ABB RAPID module: Module1.mod

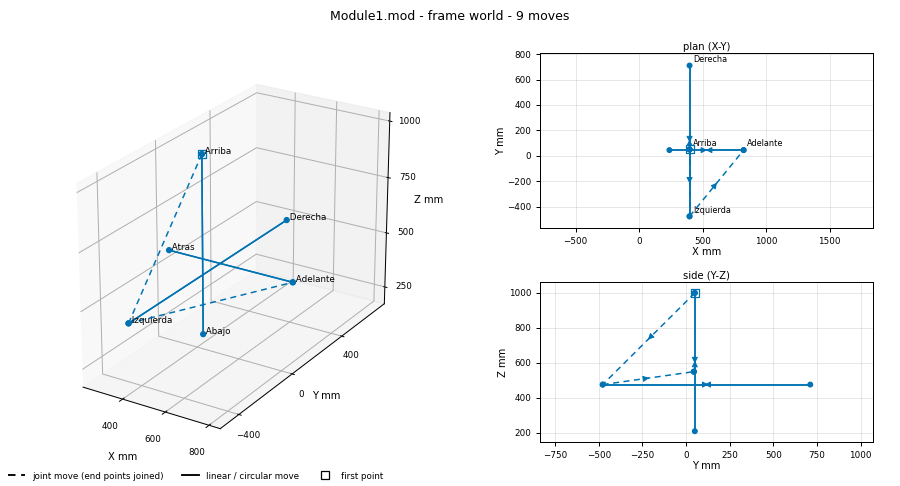
[picture p0: tool path of Module1.mod in frame world, 9 of 9 moves have a stored position in this frame; points joined in program order, loops and branches not executed]
MODULE Module1
        CONST robtarget Target_10:=[[397.237396506,49.895027971,999.967806709],[0.500000144,-0.000000762,0.86602532,-0.000000259],[0,-1,0,0],[9E+09,9E+09,9E+09,9E+09,9E+09,9E+09]];
    CONST robtarget Target_20:=[[397.2373779,49.895029997,208.416392869],[0.500000126,-0.000000768,0.866025331,-0.000000222],[0,-2,1,0],[9E+09,9E+09,9E+09,9E+09,9E+09,9E+09]];
    CONST robtarget Target_30:=[[823.141261344,44.509056663,549.297530143],[0.500000173,-0.000000339,0.866025304,-0.000000462],[0,1,-2,1],[9E+09,9E+09,9E+09,9E+09,9E+09,9E+09]];
    CONST robtarget Target_40:=[[238.396814188,44.509066911,549.297510446],[0.500000164,-0.000000322,0.866025309,-0.000000435],[0,1,-2,1],[9E+09,9E+09,9E+09,9E+09,9E+09,9E+09]];
    CONST robtarget Target_50:=[[397.237392628,-293.472887343,485.395595719],[0.500000125,-0.000000729,0.866025331,-0.000000243],[-1,0,-2,0],[9E+09,9E+09,9E+09,9E+09,9E+09,9E+09]];
    CONST robtarget Target_60:=[[397.237393587,50.453069476,485.39558546],[0.500000114,-0.000000756,0.866025338,-0.000000264],[0,1,-1,1],[9E+09,9E+09,9E+09,9E+09,9E+09,9E+09]];
    CONST robtarget Target_70:=[[802.304016355,50.453065947,615.789609831],[0.500000141,-0.000000543,0.866025322,-0.000000186],[0,1,-2,1],[9E+09,9E+09,9E+09,9E+09,9E+09,9E+09]];
    CONST robtarget Target_80:=[[271.909522335,50.453072281,615.789590887],[0.500000145,-0.000000573,0.86602532,-0.000000214],[0,1,-2,1],[9E+09,9E+09,9E+09,9E+09,9E+09,9E+09]];
    CONST robtarget Izquierda:=[[397.237378301,-477.405403417,475.381603255],[0.500000116,-0.000000746,0.866025337,-0.000000266],[-1,-2,0,1],[9E+09,9E+09,9E+09,9E+09,9E+09,9E+09]];
    CONST robtarget Derecha:=[[397.237389171,710.867878695,475.381600112],[0.500000143,-0.000000745,0.866025321,-0.000000263],[0,1,-2,1],[9E+09,9E+09,9E+09,9E+09,9E+09,9E+09]];
    CONST robtarget Arriba:=[[397.237396506,49.895027971,999.967806709],[0.500000144,-0.000000762,0.86602532,-0.000000259],[0,-1,0,0],[9E+09,9E+09,9E+09,9E+09,9E+09,9E+09]];
    CONST robtarget Abajo:=[[397.2373779,49.895029997,208.416392869],[0.500000126,-0.000000768,0.866025331,-0.000000222],[0,-2,1,0],[9E+09,9E+09,9E+09,9E+09,9E+09,9E+09]];
    CONST robtarget Adelante:=[[823.141261344,44.509056663,549.297530143],[0.500000173,-0.000000339,0.866025304,-0.000000462],[0,1,-2,1],[9E+09,9E+09,9E+09,9E+09,9E+09,9E+09]];
    CONST robtarget Atras:=[[238.396814188,44.509066911,549.297510446],[0.500000164,-0.000000322,0.866025309,-0.000000435],[0,1,-2,1],[9E+09,9E+09,9E+09,9E+09,9E+09,9E+09]];
!***********************************************************
    !
    ! Module:  Module1
    !
    ! Description:
    !   <Insert description here>
    !
    ! Author: Ramiro
    !
    ! Version: 1.0
    !
    !***********************************************************


    !***********************************************************
    !
    ! Procedure main
    !
    !   This is the entry point of your program
    !
    !***********************************************************
    PROC main()
        Singularidad_Munieca;
    ENDPROC
    PROC Singularidad_Munieca()
        MoveJ Arriba,v1000,fine,tool0\WObj:=wobj0;
        MoveL Abajo,v5000,fine,tool0\WObj:=wobj0;
        MoveL Arriba,v5000,fine,tool0\WObj:=wobj0;
        MoveJ Izquierda,v5000,fine,tool0\WObj:=wobj0;
        MoveL Derecha,v5000,fine,tool0\WObj:=wobj0;
        MoveL Izquierda,v5000,fine,tool0\WObj:=wobj0;
        MoveJ Adelante,v5000,fine,tool0\WObj:=wobj0;
        MoveL Atras,v5000,fine,tool0\WObj:=wobj0;
        MoveL Adelante,v5000,fine,tool0\WObj:=wobj0;

    ENDPROC
ENDMODULE
